{attribute addProperty BoxType "EL3773-0000-0016"}
{attribute addProperty Id "I1_STATUSAT %I*I1_STATUS_F9B4A013162"}
{attribute addProperty CRC "2958739504"}
{attribute addProperty SizeInBites "16"}
{attribute addProperty SizeInBytes "2"}
TYPE L1_Current_Samples_B05AC830 :
STRUCT
	{attribute addProperty Name "I1_STATUS"}
	I1_STATUS AT %I* : I1_STATUS_F9B4A013;
END_STRUCT
END_TYPE

(* stored: Version 1.2.0.0, ProductVersion 3.1.4024.9
   DUT L1_Current_Samples_B05AC830: Id {19d13831-52e9-4a04-b179-4d65257fdf95} *)
